FUNCTION_BLOCK PUBLIC FB_CANControl IMPLEMENTS ITF_CANControl
VAR_INPUT
END_VAR
VAR_OUTPUT
END_VAR
VAR
	rxQueue AT%I* : ST_TxRxQueue;
	txQueue AT%Q* : ST_TxRxQueue;
	i : INT;
	messageRecieved : ST_TxRxMessage;
END_VAR

IF rxQueue.rxCounter <> txQueue.rxCounter THEN
	//if we have recieved a message rxCounter is incremented by interface
	M_GetMessage();
END_IF

METHOD PUBLIC M_GetMessage : BOOL
VAR_INPUT
END_VAR
FOR i := 0 TO rxQueue.noOfMessages DO
	messageRecieved := rxQueue.messages[i];
END_FOR
txQueue.rxCounter := rxQueue.rxCounter;
END_METHOD

METHOD PUBLIC M_PushMessage : BOOL
VAR_INPUT
	messageSend : ST_TxRxMessage;
END_VAR
IF txQueue.txCounter = rxQueue.TxCounter THEN
	FOR i:=0 TO 1 DO
		txQueue.messages[i] := messageSend;
	End_for
	txQueue.noOfMessages := 1;
	txQueue.TxCounter := rxQueue.TxCounter + 1;
END_IF
END_METHOD

END_FUNCTION_BLOCK

(* stored: Version 1.1.0.1, ProductVersion 3.1.4024.11
   POU FB_CANControl: Id {b6b4773b-a627-490b-a885-78ecb679b4ff}, SpecialFunc None
   Method M_GetMessage: Id {02c3fb95-bf7e-41ee-8cee-070b95293a0e}
   Method M_PushMessage: Id {ad1aea3b-53ed-43f8-bbfd-97e7f8ab76b1} *)
